Fanuc TP program (LS listing): M_EXE11.LS

/PROG  M_EXE11	  Macro
/ATTR
OWNER		= MNEDITOR;
COMMENT		= "Manual macro11";
PROG_SIZE	= 198;
CREATE		= DATE 22-03-26  TIME 13:11:56;
MODIFIED	= DATE 30-06-22  TIME 08:31:24;
FILE_NAME	= ;
VERSION		= 0;
LINE_COUNT	= 4;
MEMORY_SIZE	= 562;
PROTECT		= READ_WRITE;
TCD:  STACK_SIZE	= 0,
      TASK_PRIORITY	= 50,
      TIME_SLICE	= 0,
      BUSY_LAMP_OFF	= 0,
      ABORT_REQUEST	= 0,
      PAUSE_REQUEST	= 0;
DEFAULT_GROUP	= 1,*,*,*,*;
CONTROL_CODE	= 00000000 00000000;
/APPL
/MN
   1:  CALL ROUTER(1) ;
   2:  DO[35:Clear of Infeed]=ON ;
   3:  DO[36:Clear of Grinder]=ON ;
   4:  DO[37:Clear of Outfeed]=ON ;
/POS
/END
